{attribute 'qualified_only'}
{attribute 'strict'}
{attribute 'to_string'}

TYPE E_Sequence :
(
	Start			:= 0,
	Done			:= 32767
);
END_TYPE

(* stored: Version 1.1.0.1
   DUT E_Sequence: Id {878266bc-be24-0265-2bd8-c0f793632c5d} *)
